PROGRAM P_Simulator
VAR
	fbCraneSimulator : FB_CraneSimulator;
END_VAR

fbCraneSimulator(
	ssMethodType := BOOL_TO_SINT(G_Simulator.bSimulatorOn),
	uDCV := G_Work.fControlOutputNormalized,
	ppbar => G_Simulator.fPistonSidePressure,
	prbar => G_Simulator.fRodSidePressure,
	xm => G_Simulator.fPistonPosition
);

// Piston Animation
G_Simulator.stPistonAnimation.pt1_y := LREAL_TO_INT(fbCraneSimulator.xm * G_Parameters.stParam.stAnimationScaling.fPistonScale);
// Boom Animation
G_Simulator.fBoomAngle := F_PistonDisplacementToBoomAngle(xCyl := fbCraneSimulator.xm);
G_Simulator.fBoomAnimation := F_BoomAnimation(
	fScale := G_Parameters.stParam.stAnimationScaling.fBoomScale,
	fBoomAngle := G_Simulator.fBoomAngle,
	fBoomLength := G_Parameters.stParam.stCraneKinematics.fBoomLength,
	fBoomTipX => G_Simulator.stBoomAnimation.pt1_x,
	fBoomTipY => G_Simulator.stBoomAnimation.pt1_y
);
G_Simulator.fBoomAngleDeg := F_RadToDeg(fRad := G_Simulator.fBoomAngle);

END_PROGRAM

(* stored: Version 1.1.0.1, ProductVersion 3.1.4024.10
   POU P_Simulator: Id {536492b7-da96-4ec3-8126-8b196493af0f}, SpecialFunc None *)
